// TwinCAT 3 PLC project PLC
// ProgramVersion: 3.1.4024.0
// libraries:
//   Tc2_Standard, * (Beckhoff Automation GmbH)
//   Tc2_System, * (Beckhoff Automation GmbH)
//   Tc3_Module, * (Beckhoff Automation GmbH)
//   VisuSymbols,3.5.10.0,System
// project tree:
//   DUTs/ stProductPos.TcDUT
//   / GlobalTextList.TcGTLO, PlcTask.TcTTO
//   GVLs/ GVL.TcGVL
//   POUs/ Control.TcPOU, MAIN.TcPOU
//   POUs/Simulation/ CameraDetection.TcPOU, ConveyorMotor.TcPOU, Simulation.TcPOU
//   VISUs/ Visualization.TcVIS, VisualizationManager.TcVMO (not stored)
// real-time tasks:
//   TASK PlcTask: cycle T#10ms, priority 20, ADS port 350

CONFIGURATION PLC
    RESOURCE PLC ON TwinCAT3
        TASK PlcTask(INTERVAL := T#10ms, PRIORITY := 20);
        PROGRAM MAIN WITH PlcTask : MAIN;
    END_RESOURCE
END_CONFIGURATION

// ---- DUTs/stProductPos.TcDUT
TYPE stProductPos :
STRUCT
	X		:	REAL;
	y		:	REAL;
END_STRUCT
END_TYPE

// ---- GVLs/GVL.TcGVL
{attribute 'qualified_only'}
VAR_GLOBAL
	ProductPresenceSensor		: BOOL;
	PostCodeSensor01			: BOOL; 
	PostCodeSensor02			: BOOL;
	PostCodeSensor03			: BOOL;
	PostCodeSensor04			: BOOL;
	InvalidPostCodesSensor		: BOOL;
	StartButton	:	BOOL;
	StopButton	:	BOOL;
	
	ConveyorMotor :	BOOL;
	SwingArm01	  : BOOL;
	SwingArm02	  : BOOL;
	SwingArm03	  : BOOL;
	SwingArm04	  : BOOL;
END_VAR

// ---- POUs/MAIN.TcPOU
PROGRAM MAIN
VAR
	Control			:	Control;
END_VAR

Simulation();

Control(StartPb	:= GVL.StartButton,
		StopPb	:= GVL.StopButton,
		PresenceSensor := GVL.ProductPresenceSensor,
		PostCodeSensor01 := GVL.PostCodeSensor01,
		PostCodeSensor02 := GVL.PostCodeSensor02,
		PostCodeSensor03 := GVL.PostCodeSensor03,
		PostCodeSensor04 := GVL.PostCodeSensor04,
		InvalidPostCodeSensor := GVL.InvalidPostCodesSensor,
		ConveyorMotorCmd => GVL.ConveyorMotor,
		Arm01Cmd => GVL.SwingArm01,
		Arm02Cmd => GVL.SwingArm02,
		Arm03Cmd => GVL.SwingArm03,
		Arm04Cmd => GVL.SwingArm04,
		);

END_PROGRAM

// ---- POUs/Control.TcPOU
FUNCTION_BLOCK Control
VAR_INPUT
	StartPb					:	BOOL;		// start pushbutton
	StopPb					:	BOOL;		// stop pushbutton
	PresenceSensor			:	BOOL;		// presence sensor at camera
	PostCodeSensor01		:	BOOL;		// presence sensor at post codes 1000-1999 container
	PostCodeSensor02		:	BOOL;		// presence sensor at post codes 2000-4999 container
	PostCodeSensor03		:	BOOL;		// presence sensor at post codes 5000-6999 container
	PostCodeSensor04		:	BOOL;		// presence sensor at post codes 7000-9999 container
	InvalidPostCodeSensor	:	BOOL;		// presence sensor at invalid post code container
END_VAR

VAR_OUTPUT
	ConveyorMotorCmd	:	BOOL;		// command for conveyor motor
	Arm01Cmd			:	BOOL;		// swing arm 01
	Arm02Cmd			:	BOOL;		// swing arm 02
	Arm03Cmd			:	BOOL;		// swing arm 03
	Arm04Cmd			:	BOOL;		// swing arm 04
	ArmScrap			:	BOOL;		// swing arm for scrap product
	
	PostCodeProducts01Count	: 	UINT;		// amount of products with post codes 1000-1999
	PostCodeProducts02Count	: 	UINT;		// amount of products with post codes 2000-4999
	PostCodeProducts03Count	: 	UINT;		// amount of products with post codes 5000-6999
	PostCodeProducts04Count	: 	UINT;		// amount of products with post codes 7000-9999
	InvalidPostCodeCount	:	UINT;		// amount of products with invalid post code
END_VAR

VAR

	SeqState			:	(IDLE, 
							  RUN, 
							  WAIT_FOR_PRODUCT, 
							  PROCESSING_CAMERA, 
							  EVALUATE_POSTCODE, 
							  STOPPED);				// sequence state	
		
	ConveyorMotor		:	ConveyorMotor;			// simulation of conveyor motor
	CameraDetect		:	CameraDetection;		// camera evaluation
	ProductCode			:	STRING;					// post code evaluated by camera
	CameraReady			:	BOOL;					
	rtProductSensor		:	R_TRIG;					// edge of product sensor detection 
	Arm					:	UINT;					// swing arm to be activated
	tonProductDeliver	:	ton;					// time between camera read and proper container
	rtPostCodeSensor01	:   R_TRIG;					// detect edge of post code product 01
	rtPostCodeSensor02	: 	R_TRIG;					// detect edge of post code product 02
	rtPostCodeSensor03	: 	R_TRIG;					// detect edge of post code product 03
	rtPostCodeSensor04	: 	R_TRIG;					// detect edge of post code product 04
	rtInvalidPostCodeSensor	: R_TRIG;				// detect edge of invalid post code product
END_VAR

(*
	FB controls transport conveyor and swing arms to place incoming products
	into proper containers according to postal code read out by vision camera.
	
	Presence Sensor : detect product presence at the camera position.
	PostCodeSensor01..04 : detect falling products with deteced post code into respective containers
    InvalidPostCodeSensor : detect falling product with invalid post code into container
*)

// FB for conveyor
ConveyorMotor(RunCmd=>ConveyorMotorCmd);

// FB for camera detection
CameraDetect(Trigger:=PresenceSensor, 
			   Code=>ProductCode, 
			   CodeReady=>CameraReady);

// cyclically evaluate amount of products of each type	   
THIS^.mProductCounters();


CASE SeqState OF
	
	IDLE:	// wait to start
		IF StartPb AND NOT StopPb THEN
			SeqState := RUN;
		END_IF
		
	RUN:// run conveyor motor
		ConveyorMotor.Start:=TRUE;
		// check if motor running
		IF ConveyorMotor.RunCmd THEN
			SeqState := WAIT_FOR_PRODUCT;
		END_IF
			
	WAIT_FOR_PRODUCT:	// wait for product presence & stop the conveyor
		rtProductSensor(CLK:=PresenceSensor);
		IF rtProductSensor.Q THEN
			ConveyorMotor.Start:=FALSE;
		END_IF
		
		// wait till conveyor stopped
		IF NOT ConveyorMotor.RunCmd THEN
			SeqState := PROCESSING_CAMERA;
		END_IF
			
	PROCESSING_CAMERA:	// conveyor stopped & read out postal code from camera  
		IF NOT CameraDetect.Busy THEN
				SeqState := EVALUATE_POSTCODE;
		END_IF
		
	EVALUATE_POSTCODE:	// evaluate the postal code and activate respective swing arm
		
		THIS^.mEvaluateCameraCode(CameraCode:=ProductCode, Arm=>Arm);
		Arm01Cmd := (Arm = 1);
		Arm02Cmd := (Arm = 2);
		Arm03Cmd := (Arm = 3);
		Arm04Cmd := (Arm = 4);
		ArmScrap := (Arm = 5);
		// delay to allow product transport into proper 
		// container with activated swing arm
		tonProductDeliver.IN := TRUE;
		ConveyorMotor.Start := TRUE;
		
		IF tonProductDeliver.Q THEN
			tonProductDeliver.IN := FALSE;
			THIS^.mResetArms();
			SeqState := RUN;
		END_IF
		
	STOPPED:	// conveyor stopped
		ConveyorMotor.Start := FALSE;
		SeqState := IDLE;

END_CASE

tonProductDeliver(PT := T#12S);

IF StopPb AND SeqState <> IDLE AND SeqState <> STOPPED THEN
	SeqState := STOPPED;
END_IF

METHOD mEvaluateCameraCode : BOOL
VAR_INPUT
	CameraCode			:	STRING;
END_VAR

VAR
	GetNum				:	UINT;
END_VAR

VAR_OUTPUT
	Arm					:	UINT;
END_VAR
(*
Check if postal code is valid i.e. starts with 'PC' and has following 4 digits
*)
IF LEN(CameraCode) = 6 THEN
	IF LEFT(CameraCode, 2) = 'PC' THEN
		GetNum := STRING_TO_UINT(MID(STR:=CameraCode, LEN:=1, POS:=3));
		
		IF GetNum = 1 THEN
			Arm := 1;
		ELSIF  GetNum >=2 AND GetNum < 5 THEN
			Arm := 2;
		ELSIF  GetNum >=5 AND GetNum < 7 THEN
			Arm := 3;
		ELSIF  GetNum >=7 AND GetNum <= 9 THEN
			Arm := 4;
		ELSE
			Arm := 5;
		END_IF
	ELSE
		Arm := 5;
	END_IF
	
ELSE
	Arm := 5;
END_IF
END_METHOD

METHOD mProductCounters : BOOL
VAR_INPUT
END_VAR
// counters for products of respective post codes
rtPostCodeSensor01(CLK := PostCodeSensor01);
rtPostCodeSensor02(CLK := PostCodeSensor02);
rtPostCodeSensor03(CLK := PostCodeSensor03);
rtPostCodeSensor04(CLK := PostCodeSensor04);
rtInvalidPostCodeSensor(CLK := InvalidPostCodeSensor);

// detect falling products into respective container
IF rtPostCodeSensor01.Q THEN
	PostCodeProducts01Count := PostCodeProducts01Count + 1;
ELSIF rtPostCodeSensor02.Q THEN
	PostCodeProducts02Count := PostCodeProducts02Count + 1;
ELSIF rtPostCodeSensor03.Q THEN
	PostCodeProducts03Count := PostCodeProducts03Count + 1;
ELSIF rtPostCodeSensor04.Q THEN
	PostCodeProducts04Count := PostCodeProducts04Count + 1;
ELSIF rtInvalidPostCodeSensor.Q THEN
	InvalidPostCodeCount := InvalidPostCodeCount + 1;
END_IF

IF rtPostCodeSensor01.Q OR
	rtPostCodeSensor02.Q OR
	rtPostCodeSensor03.Q OR
	rtPostCodeSensor04.Q OR
	rtInvalidPostCodeSensor.Q THEN
	
	tonProductDeliver.IN := FALSE;
	THIS^.mResetArms();
	SeqState := RUN;
END_IF
END_METHOD

METHOD mResetArms : BOOL
VAR_INPUT
END_VAR
Arm01Cmd := FALSE;
Arm02Cmd := FALSE;
Arm03Cmd := FALSE;
Arm04Cmd := FALSE;
ArmScrap := FALSE;
END_METHOD

END_FUNCTION_BLOCK

// ---- POUs/Simulation/ConveyorMotor.TcPOU
FUNCTION_BLOCK ConveyorMotor
VAR_INPUT
	Start			:	BOOL;
END_VAR
VAR_OUTPUT
	RunCmd			:	BOOL;
END_VAR
VAR
	tonStartTime	:	TON;
	tofStopTime		:	TOF;	
END_VAR

(*
	Simulation of conveyor motor control 
*)

tonStartTime(IN:=Start , PT:=T#300MS);
tofStopTime(IN:=Start , PT:=T#200MS);

RunCmd := tonStartTime.Q OR tofStopTime.Q;

END_FUNCTION_BLOCK

// ---- POUs/Simulation/CameraDetection.TcPOU
FUNCTION_BLOCK CameraDetection
VAR_INPUT
	Trigger			:	BOOL;		// trigger for camera read
END_VAR
VAR_OUTPUT
	Code			:	STRING;		// code read out by camera
	CodeReady		:	BOOL;		// code ready 
	Busy			:	BOOL;		// processing image
END_VAR
VAR
	ftReadCamera	:	F_TRIG;
	tpReadCamera	:	TP;
	CharCodes		:	ARRAY[0..9] OF STRING(2) := ['PC', 'PC', 'PC', 'PC', 'PC', 'PC', 'KL', 'PC', 'PC', 'CG'];
	RandCode		:	DRAND;
	RandNumber		:	DRAND;
	RandVal			:	LREAL;
	Idx				:	UINT;
	CodeNumber		:	UINT;
END_VAR

(*
	Simulation of camera read detection
	Trigger starts reading process.
	Detected code is passed as Code on FB output.
	Detected code should have XXYYYY format, where
	XX - two char alphabetical code
	YYYY - four digit number  
*)

// detect trigger and delay some time for stability
tpReadCamera(IN:=Trigger,
			  PT:=T#400MS, 
			  Q=>, 
			  ET=> );
			  
IF tpReadCamera.Q THEN
	Busy := TRUE;
	CodeReady := FALSE;
ELSE
	Busy := FALSE;
END_IF
			  
ftReadCamera(CLK:=tpReadCamera.Q);
CodeReady := FALSE;
			  
IF ftReadCamera.Q THEN
	// create XX part of the code
	RandCode(Seed:=1, Num=>RandVal);
	Idx := LIMIT(0, LREAL_TO_UINT(RandVal * 10.0) - 1, 9);
	
	// create YYYY part of the code -> max value=9999
	RandNumber(Seed:=3, Num=>RandVal);
	CodeNumber := LREAL_TO_UINT(RandVal * 10000.0) - 1;
	
	IF Idx <= 9 THEN
		Code := CONCAT(CharCodes[Idx], UINT_TO_STRING(CodeNumber));
		CodeReady := TRUE;
	END_IF
END_IF

END_FUNCTION_BLOCK

// ---- POUs/Simulation/Simulation.TcPOU
PROGRAM Simulation
VAR
	ProductPosition		:	stProductPos;
	Xoffset				:	REAL;
	Yoffset				:	REAL;
	tpSensor			: 	ARRAY[1..10] OF TP;
	Idx					: 	UINT;
END_VAR

IF NOT Main.Control.Arm01Cmd AND NOT Main.Control.Arm02Cmd AND
	NOT Main.Control.Arm03Cmd AND NOT Main.Control.Arm04Cmd AND
	NOT Main.Control.ArmScrap THEN
	Xoffset := 0.5;
END_IF

IF MAIN.Control.ConveyorMotorCmd THEN
	ProductPosition.X := ProductPosition.X + Xoffset;
	ProductPosition.Y := ProductPosition.Y + Yoffset; 
END_IF

IF ProductPosition.X > 88 AND ProductPosition.X < 97 THEN
	GVL.ProductPresenceSensor := TRUE;
ELSE 
	GVL.ProductPresenceSensor := FALSE;
END_IF

IF Main.Control.Arm01Cmd AND 
	MAIN.Control.ConveyorMotorCmd AND
    ProductPosition.X >= 200 THEN
	Xoffset := 0.0;
	Yoffset := 0.4;
	
ELSIF Main.Control.Arm02Cmd AND 
	MAIN.Control.ConveyorMotorCmd AND
    ProductPosition.X >= 300 THEN
	Xoffset := 0.0;
	Yoffset := 0.4;
	
ELSIF Main.Control.Arm03Cmd AND 
	MAIN.Control.ConveyorMotorCmd AND
    ProductPosition.X >= 400 THEN
	Xoffset := 0.0;
	Yoffset := 0.4;
	
ELSIF Main.Control.Arm04Cmd AND 
	MAIN.Control.ConveyorMotorCmd AND
    ProductPosition.X >= 500 THEN
	Xoffset := 0.0;
	Yoffset := 0.4;
	
ELSIF Main.Control.ArmScrap AND 
	MAIN.Control.ConveyorMotorCmd AND
    ProductPosition.X >= 620 THEN
	Xoffset := 0.0;
	Yoffset := 0.4;
END_IF


IF ProductPosition.Y >= 60 THEN
	ProductPosition.X := 0.0;
	ProductPosition.Y := 0.0;
	Yoffset := 0.0;
END_IF

// simulation of counting sensor
tpSensor[1](PT:=T#300MS);
tpSensor[2](PT:=T#300MS);
tpSensor[3](PT:=T#300MS);
tpSensor[4](PT:=T#300MS);
tpSensor[5](PT:=T#300MS);
GVL.PostCodeSensor01 := tpSensor[1].Q;
GVL.PostCodeSensor02 := tpSensor[2].Q;
GVL.PostCodeSensor03 := tpSensor[3].Q;
GVL.PostCodeSensor04 := tpSensor[4].Q;
GVL.InvalidPostCodesSensor := tpSensor[5].Q;

FOR Idx:= 1 TO 10 DO
	IF tpSensor[Idx].Q THEN
		tpSensor[Idx].IN := FALSE;
	END_IF
END_FOR


IF ProductPosition.Y > 45 AND 
	ProductPosition.Y < 55 AND
	Main.Control.Arm01Cmd THEN
	//GVL.PostCodeSensor01 := TRUE;
	tpSensor[1].IN := TRUE;
ELSE
	;
	//GVL.PostCodeSensor01 := FALSE;
END_IF

IF ProductPosition.Y > 45 AND 
	ProductPosition.Y < 55 AND
	Main.Control.Arm02Cmd THEN
	//GVL.PostCodeSensor02 := TRUE;
	tpSensor[2].IN := TRUE;
ELSE
	;
	//GVL.PostCodeSensor02 := FALSE;
END_IF

IF ProductPosition.Y > 45 AND 
	ProductPosition.Y < 55 AND
	Main.Control.Arm03Cmd THEN
	//GVL.PostCodeSensor03 := TRUE;
	tpSensor[3].IN := TRUE;
ELSE
	;
	//GVL.PostCodeSensor03 := FALSE;
END_IF

IF ProductPosition.Y > 45 AND 
	ProductPosition.Y < 55 AND
	Main.Control.Arm04Cmd THEN
	//GVL.PostCodeSensor04 := TRUE;
	tpSensor[4].IN := TRUE;
ELSE
	;
	//GVL.PostCodeSensor04 := FALSE;
END_IF


IF ProductPosition.Y > 45 AND 
	ProductPosition.Y < 55 AND
	Main.Control.ArmScrap THEN
	tpSensor[5].IN := TRUE;
	//GVL.InvalidPostCodesSensor := TRUE;
ELSE
	;
	//GVL.InvalidPostCodesSensor := FALSE;
END_IF

END_PROGRAM

// ---- GlobalTextList.TcGTLO
TEXTLIST GlobalTextList
  225 = '1'
  818 = 'Invalid\nPost Codes'
  68 = 'Post Codes'
  18 = 'Post Codes\n1000-1999'
  668 = 'Post Codes\n2000-4999'
  97 = 'Post Codes\n5000-6999'
  685 = 'Post Codes\n7000-9999'
  382 = 'Postal Code: %s'
  602 = 'Presence \nSensor'
  725 = 'Presence Sensor'
  328 = 'Product Sorting with Vision Camera'
  33 = 'Sensor'
  139 = 'START'
  952 = 'STOP'
  110 = 'Total: %s'
END_TEXTLIST

// ---- VISUs/Visualization.TcVIS
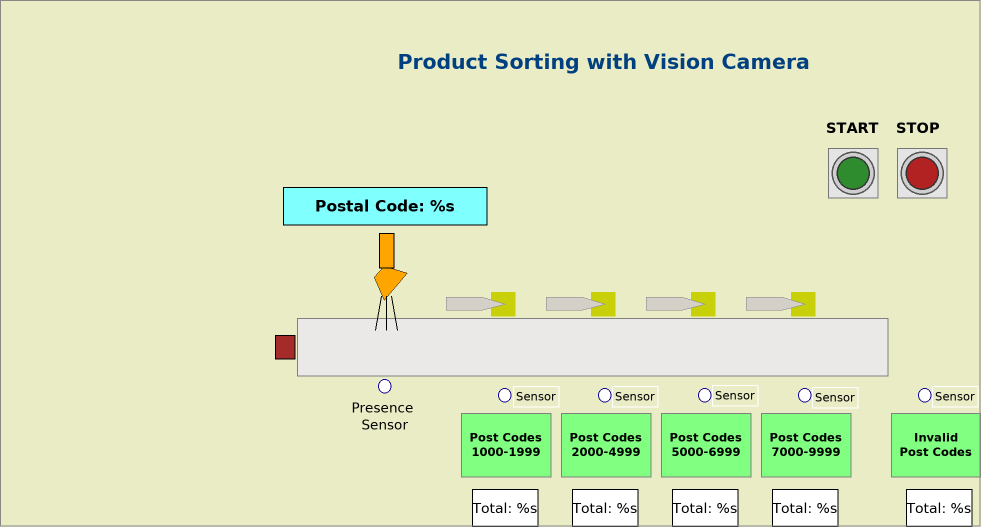
VISUALIZATION Visualization  // 981x527
    Polygon (374,277) (384,266) (407,273) (384,300), colour toggle: MAIN.Control.CameraDetect.Busy
    Rectangle (379,233 15x35)
    Rectangle (297,318 591x58), colour toggle: MAIN.Control.ConveyorMotorCmd
    Rectangle (275,335 20x24)
        p3560616238: Simulation.ProductPosition.X
        p2738717112: Simulation.ProductPosition.y
    Ellipse (378,379 13x14), colour toggle: GVL.ProductPresenceSensor
    Rectangle (491,292 24x24)
    Polygon (446,297) (482,297) (505,304) (482,310) (446,310)
        p2858320360: BOOL_TO_INT(MAIN.Control.Arm01Cmd) * 90
    Rectangle (591,292 24x24)
    Rectangle (691,292 24x24)
    Rectangle (791,292 24x24)
    Line (386,296) (386,330), invisible if: NOT MAIN.Control.CameraDetect.Busy
    Line (391,296) (397,330), invisible if: NOT MAIN.Control.CameraDetect.Busy
    Line (381,296) (375,330), invisible if: NOT MAIN.Control.CameraDetect.Busy
    Rectangle (461,413 90x64), "Post Codes 1000-1999"
    Rectangle (561,413 90x64), "Post Codes 2000-4999"
    Rectangle (661,413 90x64), "Post Codes 5000-6999"
    Rectangle (761,413 90x64), "Post Codes 7000-9999"
    Ellipse (498,388 13x14), colour toggle: GVL.PostCodeSensor01
    Rectangle (891,413 90x64), "Invalid Post Codes"
    Polygon (546,297) (582,297) (605,304) (582,310) (546,310)
        p2858320360: BOOL_TO_INT(MAIN.Control.Arm02Cmd) * 90
    Polygon (646,297) (682,297) (705,304) (682,310) (646,310)
        p2858320360: BOOL_TO_INT(MAIN.Control.Arm03Cmd) * 90
    Polygon (746,297) (782,297) (805,304) (782,310) (746,310)
        p2858320360: BOOL_TO_INT(MAIN.Control.Arm04Cmd) * 90
    Ellipse (598,388 13x14), colour toggle: GVL.PostCodeSensor02
    Ellipse (698,388 13x14), colour toggle: GVL.PostCodeSensor03
    Ellipse (798,388 13x14), colour toggle: GVL.PostCodeSensor04
    Ellipse (918,388 13x14), colour toggle: GVL.InvalidPostCodesSensor
    Rectangle (349,398 72x37), "Presence Sensor"
    Rectangle (513,386 46x21), "Sensor"
    Rectangle (612,386 46x21), "Sensor"
    Rectangle (712,385 46x21), "Sensor"
    Rectangle (812,387 46x21), "Sensor"
    Rectangle (932,386 46x21), "Sensor"
    PushSwitch (828,148 50x50), variable: GVL.StartButton, behaviour: TAP, style: Switch-PushSwitch-Green
    PushSwitch (897,148 50x50), variable: GVL.StopButton, behaviour: TAP, style: Switch-PushSwitch-Red
    RoundedRectangle (472,489 66x38), "Total: %s", text variable: MAIN.Control.PostCodeProducts01Count
    RoundedRectangle (572,489 66x38), "Total: %s", text variable: MAIN.Control.PostCodeProducts02Count
    RoundedRectangle (672,489 66x38), "Total: %s", text variable: MAIN.Control.PostCodeProducts03Count
    RoundedRectangle (772,489 66x38), "Total: %s", text variable: MAIN.Control.PostCodeProducts04Count
    RoundedRectangle (906,489 66x38), "Total: %s", text variable: MAIN.Control.InvalidPostCodeCount
    RoundedRectangle (283,187 204x38), "Postal Code: %s", text variable: MAIN.Control.ProductCode
    Rectangle (810,113 85x30), "START"
    Rectangle (885,113 66x30), "STOP"
    Rectangle (394,47 420x30), "Product Sorting with Vision Camera"
END_VISUALIZATION
